{attribute 'linkalways'} 
{attribute 'no_explicit_call' := 'This FB is a CLASS and must be accessed using methods or properties'}
{attribute 'enable_dynamic_creation'}
FUNCTION_BLOCK FINAL DIV_DWORD EXTENDS Node
VAR
	in1 : _DWORD(0);
	in2 : _DWORD(0);
	out : _DWORD(0);
	div0 : _BOOL(FALSE);
END_VAR

METHOD PUBLIC Clone : I_Node
VAR
	pNode : POINTER TO DIV_DWORD;
END_VAR
pNode := __NEW(DIV_DWORD);
Clone := pNode^;
END_METHOD

METHOD FB_init : BOOL
VAR_INPUT
	bInitRetains : BOOL; // if TRUE, the retain variables are initialized (warm start / cold start)
	bInCopyCode : BOOL;  // if TRUE, the instance afterwards gets moved into the copy code (online change)
END_VAR
AddInput('in1',THIS^.in1);
AddInput('in2',THIS^.in2);
AddOutput('out', THIS^.out);
AddOutput('div0', THIS^.div0);
END_METHOD

METHOD PROTECTED OnExecute
VAR
END_VAR
IF in2.Value = 0 THEN
	div0.Value := TRUE;
	RETURN;
END_IF

out.Value := in1.Value / in2.Value;
div0.Value := FALSE;
END_METHOD

END_FUNCTION_BLOCK

(* stored: Version 1.1.0.1, ProductVersion 3.1.4024.15
   POU DIV_DWORD: Id {f19ec0f4-8f93-44f1-8185-0521390bd989}, SpecialFunc None
   Folder Constructor: Id {4368794b-c515-4a54-b2da-4f44468ec786}
   Method Clone: Id {7a094134-e3c0-453d-85b7-b9a61edf0fb5}
   Method FB_init: Id {2f5dc07d-bde0-4ab0-97c0-1868e23a4cfc}
   Method OnExecute: Id {753121d5-1207-4f72-8ef0-7d962257b361} *)
